_CFC_ (* Continuous Function Chart, elements in execution order *)
#0 OR(SHU6_PV1_YA3_UP_RESET, SHU6_PV1_SB)
#1 SEL(SHU6_PV1_YA3_AI5_FILTER_ON, T#0ms, T#2s)
#2 fb_YA2:ISTOK_ANALOGVH(enable: TRUE, rawValue: SHU6_PV1_1YA3_AI1, reset: #0, enableLimitCtrl: TRUE, ctrlVoltage: NOT SHU6_PV1_YA3_AI5_CVOLT, changeValueWithoutPower: TRUE, highRange: YA_HIGHRANGE, lowRange: YA_LOWRANGE, highLimit: SHU6_PV1_YA_HIGHLIMIT, lowLimit: SHU6_PV1_YA_LOWLIMIT, filterTime: #1, offset: ofset, delayEnable: YA_DELAY)
#3 SHU6_PV1_YA3_UP_VN <= #2.presentValue
#4 SHU6_PV1_YA3_UP_DOST <= #2.reliability
#5 Lt_otkr_zakr:ISTOK_LT(dost: #2.reliability, x: #2.presentValue, ust: 5, shkal: -, gist: 3)
#6 SHU6_PV1_YA3_ZKR <= #5.Xm
#7 gt_otkr_otr:ISTOK_GT(dost: #2.reliability, x: #2.presentValue, ust: 95, shkal: -, gist: 3)
#8 SHU6_PV1_YA3_OTK <= #7.Xb
#9 SUB(YA3_UST_VKL_STER_REG, YA3_UST_OTKL_STER_REG)
#10 fb_YA2bUST_VKL_STER_REG:ISTOK_GT(dost: #2.reliability, x: #2.presentValue, ust: YA3_UST_VKL_STER_REG, shkal: -, gist: #9)
#11 SHU6_PV1_YA3_B_UST_VKL_STER_REG <= #10.Xb
#12 SHU6_PV1_YA3_M_UST_VKL_STER_REG <= #10.XbN
#13 SUB(YA3_UST_OTKL_UVEL_CHAST, YA3_UST_VKL_UVEL_CHAST)
#14 fb_YA2mOTKL_STER_REG:ISTOK_LT(dost: #2.reliability, x: #2.presentValue, ust: YA3_UST_VKL_UVEL_CHAST, shkal: -, gist: #13)
#15 SHU6_PV1_YA3_M_UST_VKL_UVEL_CHAST <= #14.Xm
#16 SHU6_PV1_YA3_B_UST_VKL_UVEL_CHAST <= #14.XmN
_END_CFC_
(* the same logic as Structured Text *)
fb_YA2(enable := TRUE, rawValue := SHU6_PV1_1YA3_AI1, reset := SHU6_PV1_YA3_UP_RESET OR SHU6_PV1_SB, enableLimitCtrl := TRUE, ctrlVoltage := NOT SHU6_PV1_YA3_AI5_CVOLT, changeValueWithoutPower := TRUE, highRange := YA_HIGHRANGE, lowRange := YA_LOWRANGE, highLimit := SHU6_PV1_YA_HIGHLIMIT, lowLimit := SHU6_PV1_YA_LOWLIMIT, filterTime := SEL(SHU6_PV1_YA3_AI5_FILTER_ON, T#0ms, T#2s), offset := ofset, delayEnable := YA_DELAY);
SHU6_PV1_YA3_UP_VN := fb_YA2.presentValue;
SHU6_PV1_YA3_UP_DOST := fb_YA2.reliability;
Lt_otkr_zakr(dost := fb_YA2.reliability, x := fb_YA2.presentValue, ust := 5, gist := 3);
SHU6_PV1_YA3_ZKR := Lt_otkr_zakr.Xm;
gt_otkr_otr(dost := fb_YA2.reliability, x := fb_YA2.presentValue, ust := 95, gist := 3);
SHU6_PV1_YA3_OTK := gt_otkr_otr.Xb;
fb_YA2bUST_VKL_STER_REG(dost := fb_YA2.reliability, x := fb_YA2.presentValue, ust := YA3_UST_VKL_STER_REG, gist := YA3_UST_VKL_STER_REG - YA3_UST_OTKL_STER_REG);
SHU6_PV1_YA3_B_UST_VKL_STER_REG := fb_YA2bUST_VKL_STER_REG.Xb;
SHU6_PV1_YA3_M_UST_VKL_STER_REG := fb_YA2bUST_VKL_STER_REG.XbN;
fb_YA2mOTKL_STER_REG(dost := fb_YA2.reliability, x := fb_YA2.presentValue, ust := YA3_UST_VKL_UVEL_CHAST, gist := YA3_UST_OTKL_UVEL_CHAST - YA3_UST_VKL_UVEL_CHAST);
SHU6_PV1_YA3_M_UST_VKL_UVEL_CHAST := fb_YA2mOTKL_STER_REG.Xm;
SHU6_PV1_YA3_B_UST_VKL_UVEL_CHAST := fb_YA2mOTKL_STER_REG.XmN;
END_PROGRAM

(* POU Input/AI/YA4_POS, CFC *)
PROGRAM YA4_POS
VAR
	fb_YA3: ISTOK_ANALOGVH;
	ofset: REAL;
	Lt_otkr_zakr: ISTOK_LT;
	gt_otkr_otr: ISTOK_GT;
	fb_YA3bUST_VKL_STER_REG: ISTOK_GT;
	fb_YA3mOTKL_STER_REG: ISTOK_LT;
END_VAR
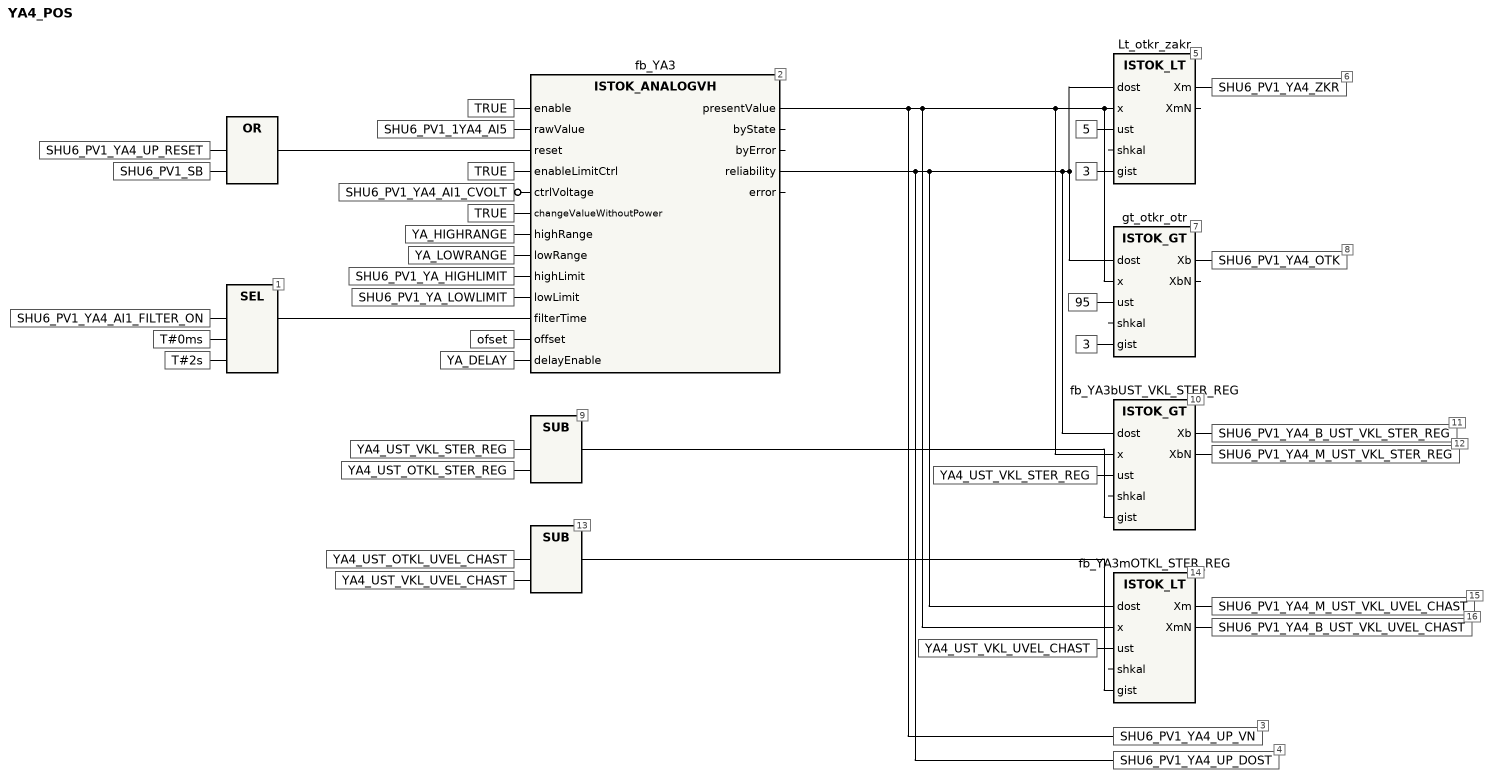
